// TIA Portal V19 export
DATA_BLOCK "DriveDiagInterfaceHmi"   // DB46
TITLE = DriveDiagInterfaceHmi
AUTHOR : Siemens Digital Industries
FAMILY : LAF
NAME : LAF_DriveDiagInterfaceHmi
VERSION : 1.1
// HMI interface for drive diagnostic
// stored: MemoryReserve 100
   VAR
      diagStatus : "LAF_typeDriveDiagInterfaceHmi";
   END_VAR
BEGIN
END_DATA_BLOCK
